{attribute 'strict'}
TYPE EFeedbackMsgStage :
(
	PositionMsg := 10
);
END_TYPE

(* stored: Version 1.1.0.1, ProductVersion 3.1.4024.12
   DUT EFeedbackMsgStage: Id {83097092-0c29-4376-a28e-c35b865c703e} *)
